INTERFACE I_Velocity

PROPERTY InVelocity : BOOL
GET
END_GET
END_PROPERTY

METHOD MoveAtVelocity : HRESULT
VAR_INPUT
	Direction : MC_Direction;
	Velocity : MC_LREAL;
END_VAR
END_METHOD

END_INTERFACE

(* stored: Version 1.1.0.1
   Itf I_Velocity: Id {bdeea844-06c8-4676-b25f-b2c6e73485b3}
   Property InVelocity: Id {e46b6806-c48d-4c44-a307-8df8a0a2793a}
   Get Get: Id {0a0bb234-8e53-4082-a9af-400da8059b8c}
   Method MoveAtVelocity: Id {56b7b37d-76b7-4396-9126-21e2fa4df7b0} *)
